// TIA Portal V20 export
TYPE "LER_typeStatusEm4"
// stored: Access Published
   STRUCT
      anodePnP1XCamEnabled : Bool;
      anodePnP1ZCamEnabled : Bool;
      anodePnP2XCamEnabled : Bool;
      anodePnP2ZCamEnabled : Bool;
      anodeDownComplete1 : Bool;
      anodeDownComplete2 : Bool;
      anodeSupplyCheck : Bool;
      anodeFinishCheck : Bool;
      anodeSupplyComplete : Bool;
      anodeFinishComplete : Bool;
      anodeReady : Bool;
      anodeRequest : Bool;
      stackJobCompleteChecked : Bool;
      stopRequest : Bool;
      stopComplete : Bool;
      anodePnP1HomePos : Bool;
      anodePnP1WorkPos : Bool;
      anodePnP2HomePos : Bool;
      anodePnP2WorkPos : Bool;
      anodeAvoidPos : Bool;
      anodeReelcutRequest : Bool;
      anodeStartCase : DInt;
      anodePnPXStart : LReal := 0.0;
      anodePnPXEnd : LReal := 75.0;
      anodePnPZDownStart : LReal := 65.0;
      anodePnPZDownEnd : LReal := 75.0;
      anodePnPZUpStart : LReal := 90.0;
      anodePnPZUpEnd : LReal := 100.0;
      anodePnP1ZOnPos : LReal := 5.0;
      anodePnP1ZOffPos : LReal := 5.0;
      anodeReelCutOnPos : LReal := 5.0;
      anodePnP2ZOnPos : LReal := 5.0;
      anodePnP2ZOffPos : LReal := 5.0;
      anodeAlignOnPos : LReal := 5.0;
      anodeAlignOffPos : LReal := 5.0;
      anodeVisionTrigger : LReal := 5.0;
      anodeVisionClean : LReal := 5.0;
   END_STRUCT;
END_TYPE
